FUNCTION_BLOCK FB_3eTI_iMesh_GasSensor EXTENDS FB_3eTI_iMesh_Base
VAR_INPUT
END_VAR
VAR_OUTPUT
END_VAR
VAR
	A 		: LREAL := 75;
	Tau 	: LREAL := 0.5;
	PV		: LREAL := 0.0;
	tk		: LREAL := 0.0;
	deltaT	:LREAL 	:= 10E-3;
	Pch     : LREAL := 10;
	remk: LREAL := 0.0;
END_VAR


// XMEAS RANGES
G_PARAMS.A_FLOW_MAX 	:=A;
G_PARAMS.D_FLOW_MAX		:=A;
G_PARAMS.E_FLOW_MAX		:=A;
G_PARAMS.AC_FLOW_MAX	:=A;

G_PARAMS.A_FLOW_MIN 	:=0.0;
G_PARAMS.D_FLOW_MIN		:=0.0;
G_PARAMS.E_FLOW_MIN		:=0.0;
G_PARAMS.AC_FLOW_MIN	:=0.0;

(* For built-in PV generator
// gas influx variables
tk := tk + deltaT;
remk := lmod(tk,2*Pch);
IF remk < Pch THEN
	PV := A*(1-EXP(-Tau*remk));
ELSE
	PV := A*EXP(-Tau*(remk-pch));
END_IF

G_IO.XMEAS[1] := PV;
G_IO.XMEAS[2] := PV;
G_IO.XMEAS[3] := PV;
G_IO.XMEAS[4] := PV;
*)

// execute the signal conversion
SUPER^();

END_FUNCTION_BLOCK

(* stored: Version 1.1.0.1, ProductVersion 3.1.4020.12
   POU FB_3eTI_iMesh_GasSensor: Id {79745510-0645-48ed-8e8c-3995314f7dfb}, SpecialFunc None *)
